// TIA Portal V20 export
FUNCTION_BLOCK "LER_EnableDisable_CM_AxisCtrl"   // FB195, LAD
// stored: Access Published, MemoryReserve 100, SetENOAutomatically false
   VAR_INPUT
      UnitStatus_mode : "LUC_typeModes";
      UnitStatus_state : "LUC_typeStates";
      emFeedBackisLinked : Bool;
      Emnodes_slmPowerMcOff : Bool;
      Emnodes_slmPowerMcRun : Bool;
      Enabletimeinterlock_afterprodmode : Bool;
      MainOpMode : "LWONIK_typeOperationMode";
      doorOpenRequest : Bool;
   END_VAR
   VAR_OUTPUT
      axisEnableCmd : Bool;
      axisEnabledMonitoring : Bool;
   END_VAR
   VAR_IN_OUT
      CmControlNode : "LBC_typeAxisControlNode";
      CmModuleInterface : "LBC_typeAxisControlInterface";
   END_VAR
   VAR
      statPulse1 : Bool;
      statpulse2 : Bool;
      statpulse3 : Bool;
      statpulse4 : Bool;
      statpulse5 : Bool;
      statpulse6 : Bool;
      statpulse7 : Bool;
      statpulse8 : Bool;
      statpulse9 : Bool;
      statpulse10 : Bool;
      statTrigger1 : Bool;
      statTrigger2 : Bool;
   END_VAR
   VAR_TEMP   // added for the SCL form of the ladder/FBD networks
      _w1 : Bool;
   END_VAR
BEGIN

REGION Network 1: Set axis enable
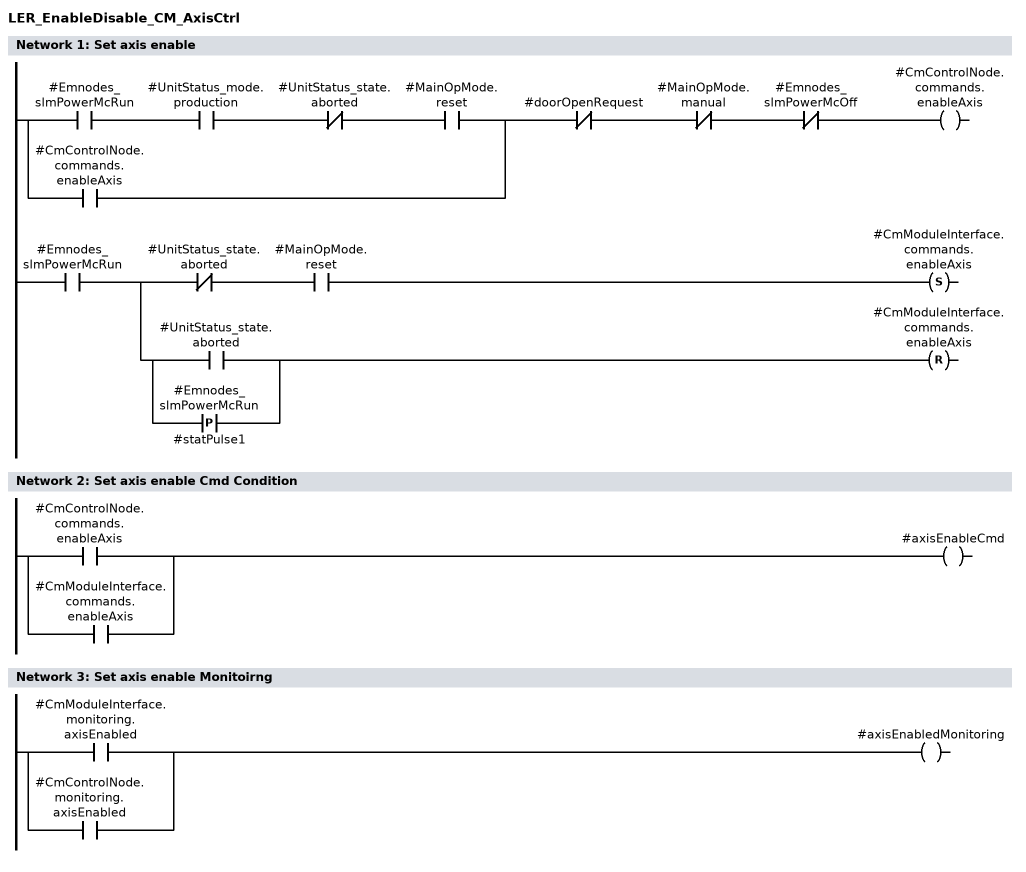
   RUNG wire#powerrail
      Contact( #Emnodes_slmPowerMcRun )
      Contact( #UnitStatus_mode.production )
      I_Contact( #UnitStatus_state.aborted )
      Contact( #MainOpMode.reset )
      wire#w1
      I_Contact( #doorOpenRequest )
      I_Contact( #MainOpMode.manual )
      I_Contact( #Emnodes_slmPowerMcOff )
      Coil( #CmControlNode.commands.enableAxis )
   END_RUNG
   RUNG wire#powerrail
      Contact( #CmControlNode.commands.enableAxis )
   END_RUNG wire#w1
   RUNG wire#powerrail
      Contact( #Emnodes_slmPowerMcRun )
      wire#w2
      I_Contact( #UnitStatus_state.aborted )
      Contact( #MainOpMode.reset )
      S_Coil( #CmModuleInterface.commands.enableAxis )
   END_RUNG
   RUNG wire#w2
      Contact( #UnitStatus_state.aborted )
      wire#w3
      R_Coil( #CmModuleInterface.commands.enableAxis )
   END_RUNG
   RUNG wire#w2
      P_Contact(operand := #Emnodes_slmPowerMcRun, bit := #statPulse1)
   END_RUNG wire#w3
   // the same network as SCL:
   #CmControlNode.commands.enableAxis := ((#Emnodes_slmPowerMcRun AND #UnitStatus_mode.production AND NOT #UnitStatus_state.aborted AND #MainOpMode.reset) OR #CmControlNode.commands.enableAxis) AND NOT #doorOpenRequest AND NOT #MainOpMode.manual AND NOT #Emnodes_slmPowerMcOff;
   IF #Emnodes_slmPowerMcRun AND NOT #UnitStatus_state.aborted AND #MainOpMode.reset THEN
       #CmModuleInterface.commands.enableAxis := TRUE;
   END_IF;
   #_w1 := #Emnodes_slmPowerMcRun AND #Emnodes_slmPowerMcRun AND NOT #statPulse1;   // rising edge of #Emnodes_slmPowerMcRun
   #statPulse1 := #Emnodes_slmPowerMcRun;
   IF (#Emnodes_slmPowerMcRun AND #UnitStatus_state.aborted) OR #_w1 THEN
       #CmModuleInterface.commands.enableAxis := FALSE;
   END_IF;
END_REGION

REGION Network 2: Set axis enable Cmd Condition
   RUNG wire#powerrail
      Contact( #CmControlNode.commands.enableAxis )
      wire#w1
      Coil( #axisEnableCmd )
   END_RUNG
   RUNG wire#powerrail
      Contact( #CmModuleInterface.commands.enableAxis )
   END_RUNG wire#w1
   // the same network as SCL:
   #axisEnableCmd := #CmControlNode.commands.enableAxis OR #CmModuleInterface.commands.enableAxis;
END_REGION

REGION Network 3: Set axis enable Monitoirng
   RUNG wire#powerrail
      Contact( #CmModuleInterface.monitoring.axisEnabled )
      wire#w1
      Coil( #axisEnabledMonitoring )
   END_RUNG
   RUNG wire#powerrail
      Contact( #CmControlNode.monitoring.axisEnabled )
   END_RUNG wire#w1
   // the same network as SCL:
   #axisEnabledMonitoring := #CmModuleInterface.monitoring.axisEnabled OR #CmControlNode.monitoring.axisEnabled;
END_REGION
END_FUNCTION_BLOCK
